Staubli VAL3: exo11.pgx

program exo11()
begin
  movej(jdepart,tstylo,mlent)
  movej(ppa,tstylo,mlent)
  movej(ppb,tstylo,mlent)
  movej(ppc,tstylo,mlent)
  movej(ppd,tstylo,mlent)
  movej(ppe,tstylo,mlent)
  movej(ppa,tstylo,mlent)
  movej(jdepart,tstylo,mlent)
  waitEndMove()
end
